// TIA Portal V20 export
TYPE "LER_typePLCToMotion"
// stored: Access Published
   STRUCT
      Commands : Struct
         Dancer : Struct
            Enable : Bool;
            Stop : Bool;
            Reset : Bool;
         END_STRUCT;
         StackMain : Struct
            Calculate : Bool;
            SemiStep : Bool;
            FullStep : Bool;
            Auto : Bool;
            SepaClean : Bool;
            CycleStop : Bool;
            FastStop : Bool;
            Reset : Bool;
         END_STRUCT;
      END_STRUCT;
      Parameters : Struct
         Dancer : Struct
            DancerDirection : Bool;
            UnWinderDirection : Bool;
            UnwinderTopUse : Bool;
            UnwinderBottomUse : Bool;
            Setpoint : LReal;
            Input : LReal;
            Kp : LReal;
            Ki : LReal;
            Radius : LReal;
            JogMode : Bool;
         END_STRUCT;
         StackMain : Struct
            Global : Struct
               CPM : LReal;
               StageWidth : LReal;
            END_STRUCT;
            "Step" : Struct
               MandrelUse : Bool;
               InitialPosFinalRoller : LReal;
               InitialPosCompensator : LReal;
            END_STRUCT;
            Auto : Struct
               SepaClean : Bool;
               CellCount : DInt;
               InitialPosFinalRoller : LReal;
               InitialPosCompensator : LReal;
               InitialPosAnodePnPX1 : LReal;
               InitialPosAnodePnPX2 : LReal;
               InitialPosAnodePnPZ1 : LReal;
               InitialPosAnodePnPZ2 : LReal;
               InitialPosCathodePnPX1 : LReal;
               InitialPosCathodePnPX2 : LReal;
               InitialPosCathodePnPZ1 : LReal;
               InitialPosCathodePnPZ2 : LReal;
               InitialPosAnodeMandrelYFront : LReal;
               InitialPosAnodeMandrelYRear : LReal;
               InitialPosAnodeMandrelZFront : LReal;
               InitialPosAnodeMandrelZRear : LReal;
               InitialPosCathodeMandrelYFront : LReal;
               InitialPosCathodeMandrelYRear : LReal;
               InitialPosCathodeMandrelZFront : LReal;
               InitialPosCathodeMandrelZRear : LReal;
               Pos1FinalRollerXFwdOutputCam : LReal;
               Pos1FinalRollerXBwdOutputCam : LReal;
               Pos1FinalRollerXStackTableDownOutputCam : LReal;
               Pos1FinalRollerXStackAnodeVisionOutputCam : LReal;
               Pos1FinalRollerXStackCathodeVisionOutputCam : LReal;
               Pos1AnodePnPX1FwdOutputCam : LReal;
               Pos1AnodePnPX1BwdOutputCam : LReal;
               Pos1AnodePnPX1ReelCutDataDeleteOffOutputCam : LReal;
               Pos1AnodePnPX2FwdOutputCam : LReal;
               Pos1AnodePnPX2BwdOutputCam : LReal;
               Pos1AnodePnPZ1Down1OutputCam : LReal;
               Pos1AnodePnPZ1Up1OutputCam : LReal;
               Pos1AnodePnPZ2Down1OutputCam : LReal;
               Pos1AnodePnPZ2Up1OutputCam : LReal;
               Pos1AnodePnPZ1Down2OutputCam : LReal;
               Pos1AnodePnPZ1Up2OutputCam : LReal;
               Pos1AnodePnPZ2Down2OutputCam : LReal;
               Pos1AnodePnPZ2Up2OutputCam : LReal;
               Pos1AnodePnPZ1SuctionOnOutputCam : LReal;
               Pos1AnodePnPZ1SuctionOffOutputCam : LReal;
               Pos1AnodePnPZ1ReelCutBlowOutputCam : LReal;
               Pos1AnodePnPZ1ReelCutDataDeleteOnOutputCam : LReal;
               Pos1AnodePnPZ1AlignVisionOutputCam : LReal;
               Pos1AnodePnPZ2SuctionOnOutputCam : LReal;
               Pos1AnodePnPZ2SuctionOffOutputCam : LReal;
               Pos1AnodeAlignSuctionOnOutputCam : LReal;
               Pos1AnodeAlignSuctionOffOutputCam : LReal;
               Pos1CathodePnPX1FwdOutputCam : LReal;
               Pos1CathodePnPX1BwdOutputCam : LReal;
               Pos1CathodePnPX1ReelCutDataDeleteOffOutputCam : LReal;
               Pos1CathodePnPX2FwdOutputCam : LReal;
               Pos1CathodePnPX2BwdOutputCam : LReal;
               Pos1CathodePnPZ1Down1OutputCam : LReal;
               Pos1CathodePnPZ1Up1OutputCam : LReal;
               Pos1CathodePnPZ2Down1OutputCam : LReal;
               Pos1CathodePnPZ2Up1OutputCam : LReal;
               Pos1CathodePnPZ1Down2OutputCam : LReal;
               Pos1CathodePnPZ1Up2OutputCam : LReal;
               Pos1CathodePnPZ2Down2OutputCam : LReal;
               Pos1CathodePnPZ2Up2OutputCam : LReal;
               Pos1CathodePnPZ1SuctionOnOutputCam : LReal;
               Pos1CathodePnPZ1SuctionOffOutputCam : LReal;
               Pos1CathodePnPZ1ReelCutBlowOutputCam : LReal;
               Pos1CathodePnPZ1ReelCutDataDeleteOnOutputCam : LReal;
               Pos1CathodePnPZ1AlignVisionOutputCam : LReal;
               Pos1CathodePnPZ2SuctionOnOutputCam : LReal;
               Pos1CathodePnPZ2SuctionOffOutputCam : LReal;
               Pos1CathodeAlignSuctionOnOutputCam : LReal;
               Pos1CathodeAlignSuctionOffOutputCam : LReal;
               Pos2FinalRollerXFwdOutputCam : LReal;
               Pos2FinalRollerXBwdOutputCam : LReal;
               Pos2FinalRollerXStackTableDownOutputCam : LReal;
               Pos2FinalRollerXStackAnodeVisionOutputCam : LReal;
               Pos2FinalRollerXStackCathodeVisionOutputCam : LReal;
               Pos2AnodePnPX1FwdOutputCam : LReal;
               Pos2AnodePnPX1BwdOutputCam : LReal;
               Pos2AnodePnPX1ReelCutDataDeleteOffOutputCam : LReal;
               Pos2AnodePnPX2FwdOutputCam : LReal;
               Pos2AnodePnPX2BwdOutputCam : LReal;
               Pos2AnodePnPZ1Down1OutputCam : LReal;
               Pos2AnodePnPZ1Up1OutputCam : LReal;
               Pos2AnodePnPZ2Down1OutputCam : LReal;
               Pos2AnodePnPZ2Up1OutputCam : LReal;
               Pos2AnodePnPZ1Down2OutputCam : LReal;
               Pos2AnodePnPZ1Up2OutputCam : LReal;
               Pos2AnodePnPZ2Down2OutputCam : LReal;
               Pos2AnodePnPZ2Up2OutputCam : LReal;
               Pos2AnodePnPZ1SuctionOnOutputCam : LReal;
               Pos2AnodePnPZ1SuctionOffOutputCam : LReal;
               Pos2AnodePnPZ1ReelCutBlowOutputCam : LReal;
               Pos2AnodePnPZ1ReelCutDataDeleteOnOutputCam : LReal;
               Pos2AnodePnPZ1AlignVisionOutputCam : LReal;
               Pos2AnodePnPZ2SuctionOnOutputCam : LReal;
               Pos2AnodePnPZ2SuctionOffOutputCam : LReal;
               Pos2AnodeAlignSuctionOnOutputCam : LReal;
               Pos2AnodeAlignSuctionOffOutputCam : LReal;
               Pos2CathodePnPX1FwdOutputCam : LReal;
               Pos2CathodePnPX1BwdOutputCam : LReal;
               Pos2CathodePnPX1ReelCutDataDeleteOffOutputCam : LReal;
               Pos2CathodePnPX2FwdOutputCam : LReal;
               Pos2CathodePnPX2BwdOutputCam : LReal;
               Pos2CathodePnPZ1Down1OutputCam : LReal;
               Pos2CathodePnPZ1Up1OutputCam : LReal;
               Pos2CathodePnPZ2Down1OutputCam : LReal;
               Pos2CathodePnPZ2Up1OutputCam : LReal;
               Pos2CathodePnPZ1Down2OutputCam : LReal;
               Pos2CathodePnPZ1Up2OutputCam : LReal;
               Pos2CathodePnPZ2Down2OutputCam : LReal;
               Pos2CathodePnPZ2Up2OutputCam : LReal;
               Pos2CathodePnPZ1SuctionOnOutputCam : LReal;
               Pos2CathodePnPZ1SuctionOffOutputCam : LReal;
               Pos2CathodePnPZ1ReelCutBlowOutputCam : LReal;
               Pos2CathodePnPZ1ReelCutDataDeleteOnOutputCam : LReal;
               Pos2CathodePnPZ1AlignVisionOutputCam : LReal;
               Pos2CathodePnPZ2SuctionOnOutputCam : LReal;
               Pos2CathodePnPZ2SuctionOffOutputCam : LReal;
               Pos2CathodeAlignSuctionOnOutputCam : LReal;
               Pos2CathodeAlignSuctionOffOutputCam : LReal;
            END_STRUCT;
            StackCalculate : Struct
               Direction : Bool := TRUE;
               RatioOption : Bool := TRUE;
               TimeOption : Bool;
               PosOption : Bool;
               DoubleOption : Bool;
               StageHeight : LReal := 360.0;
               StageGap : LReal := 5.0;
               AccRatio : DInt := 3;
               Ratio : Struct
                  FinalRollerStart : LReal := 0.0;
                  FinalRollerEnd : LReal := 75.0;
                  PnPXStart : LReal := 0.0;
                  PnPXEnd : LReal := 75.0;
                  PnPZDownStart : LReal := 65.0;
                  PnPZDownEnd : LReal := 75.0;
                  PnPZUpStart : LReal := 90.0;
                  PnPZUpEnd : LReal := 100.0;
                  MandrelBwdStart : LReal := 75.0;
                  MandrelBwdEnd : LReal := 82.5;
                  MandrelFwdStart : LReal := 82.5;
                  MandrelFwdEnd : LReal := 90.0;
                  MandrelUpStart1 : LReal := 55.0;
                  MandrelUpEnd1 : LReal := 62.5;
                  MandrelUpStart2 : LReal := 75.0;
                  MandrelUpEnd2 : LReal := 82.5;
                  MandrelDownStart : LReal := 87.0;
                  MandrelDownEnd : LReal := 90.0;
                  MandrelYTerm : LReal := 0.0;
                  MandrelZTerm : LReal := 0.0;
                  MandrelBwdOffset : LReal := 0.0;
                  MandrelFwdOffset : LReal := 0.0;
               END_STRUCT;
               "Time" : Struct
                  FinalRollerStart : LReal;
                  FinalRollerEnd : LReal;
                  PnPXStart : LReal;
                  PnPXEnd : LReal;
                  PnPZDownStart : LReal;
                  PnPZDownEnd : LReal;
                  PnPZUpStart : LReal;
                  PnPZUpEnd : LReal;
                  MandrelBwdStart : LReal;
                  MandrelBwdEnd : LReal;
                  MandrelFwdStart : LReal;
                  MandrelFwdEnd : LReal;
                  MandrelUpStart1 : LReal;
                  MandrelUpEnd1 : LReal;
                  MandrelUpStart2 : LReal;
                  MandrelUpEnd2 : LReal;
                  MandrelDownStart : LReal;
                  MandrelDownEnd : LReal;
               END_STRUCT;
               Position : Struct
                  FinalRollerBwdPos : LReal;
                  FinalRollerFwdPos : LReal;
               END_STRUCT;
               TeachingPos : Struct
                  StartPos : Struct
                     Compensator : LReal;
                     FinalRoller : LReal;
                     AnodePnPX1 : LReal;
                     AnodePnPX2 : LReal;
                     AnodePnPZ1 : LReal;
                     AnodePnPZ2 : LReal;
                     CathodePnPX1 : LReal;
                     CathodePnPX2 : LReal;
                     CathodePnPZ1 : LReal;
                     CathodePnPZ2 : LReal;
                     AnodeMandrelYFront : LReal;
                     AnodeMandrelYRear : LReal;
                     AnodeMandrelZFront : LReal;
                     AnodeMandrelZRear : LReal;
                     CathodeMandrelYFront : LReal;
                     CathodeMandrelYRear : LReal;
                     CathodeMandrelZFront : LReal;
                     CathodeMandrelZRear : LReal;
                  END_STRUCT;
                  EndPos : Struct
                     FinalRoller : LReal;
                     AnodePnPX1 : LReal;
                     AnodePnPX2 : LReal;
                     AnodePnPZ1P1 : LReal;
                     AnodePnPZ1P2 : LReal;
                     AnodePnPZ2P1 : LReal;
                     AnodePnPZ2P2 : LReal;
                     CathodePnPX1 : LReal;
                     CathodePnPX2 : LReal;
                     CathodePnPZ1P1 : LReal;
                     CathodePnPZ1P2 : LReal;
                     CathodePnPZ2P1 : LReal;
                     CathodePnPZ2P2 : LReal;
                     AnodeMandrelYFront : LReal;
                     AnodeMandrelYRear : LReal;
                     AnodeMandrelZFront : LReal;
                     AnodeMandrelZRear : LReal;
                     CathodeMandrelYFront : LReal;
                     CathodeMandrelYRear : LReal;
                     CathodeMandrelZFront : LReal;
                     CathodeMandrelZRear : LReal;
                  END_STRUCT;
               END_STRUCT;
            END_STRUCT;
         END_STRUCT;
      END_STRUCT;
      TechnologyObject : Struct
         Axis : Struct
            MasterVirtual : DB_ANY := 85;
            UnwinderVirtual : DB_ANY := 391;
            UnwinderTop : DB_ANY := 364;
            UnwinderBottom : DB_ANY := 263;
            FinalRoller : DB_ANY := 171;
            Compensator : DB_ANY := 143;
            AnodePnPX1 : DB_ANY := 144;
            AnodePnPX2 : DB_ANY := 145;
            AnodePnPZ1 : DB_ANY := 149;
            AnodePnPZ2 : DB_ANY := 150;
            CathodePnPX1 : DB_ANY := 146;
            CathodePnPX2 : DB_ANY := 147;
            CathodePnPZ1 : DB_ANY := 151;
            CathodePnPZ2 : DB_ANY := 153;
            AnodeMandrelYFront : DB_ANY := 163;
            AnodeMandrelYRear : DB_ANY := 162;
            AnodeMandrelZFront : DB_ANY := 167;
            AnodeMandrelZRear : DB_ANY := 166;
            CathodeMandrelYFront : DB_ANY := 161;
            CathodeMandrelYRear : DB_ANY := 160;
            CathodeMandrelZFront : DB_ANY := 165;
            CathodeMandrelZRear : DB_ANY := 164;
            SepaClampX : DB_ANY := 178;
         END_STRUCT;
         Cam : Struct
            FinalRollerCam { ExternalAccessible := 'False'; ExternalVisible := 'False'; ExternalWritable := 'False'} : DB_ANY := 281;
            CompensatorCam { ExternalAccessible := 'False'; ExternalVisible := 'False'; ExternalWritable := 'False'} : DB_ANY := 69;
            AnodePnPX1Cam { ExternalAccessible := 'False'; ExternalVisible := 'False'; ExternalWritable := 'False'} : DB_ANY := 230;
            AnodePnPX2Cam { ExternalAccessible := 'False'; ExternalVisible := 'False'; ExternalWritable := 'False'} : DB_ANY := 295;
            AnodePnPZ1Cam { ExternalAccessible := 'False'; ExternalVisible := 'False'; ExternalWritable := 'False'} : DB_ANY := 294;
            AnodePnPZ2Cam { ExternalAccessible := 'False'; ExternalVisible := 'False'; ExternalWritable := 'False'} : DB_ANY := 296;
            CathodePnPX1Cam { ExternalAccessible := 'False'; ExternalVisible := 'False'; ExternalWritable := 'False'} : DB_ANY := 293;
            CathodePnPX2Cam { ExternalAccessible := 'False'; ExternalVisible := 'False'; ExternalWritable := 'False'} : DB_ANY := 297;
            CathodePnPZ1Cam { ExternalAccessible := 'False'; ExternalVisible := 'False'; ExternalWritable := 'False'} : DB_ANY := 299;
            CathodePnPZ2Cam { ExternalAccessible := 'False'; ExternalVisible := 'False'; ExternalWritable := 'False'} : DB_ANY := 298;
            AnodeMandrelYFrontCam { ExternalAccessible := 'False'; ExternalVisible := 'False'; ExternalWritable := 'False'} : DB_ANY := 283;
            AnodeMandrelYRearCam { ExternalAccessible := 'False'; ExternalVisible := 'False'; ExternalWritable := 'False'} : DB_ANY := 285;
            AnodeMandrelZFrontCam { ExternalAccessible := 'False'; ExternalVisible := 'False'; ExternalWritable := 'False'} : DB_ANY := 287;
            AnodeMandrelZRearCam { ExternalAccessible := 'False'; ExternalVisible := 'False'; ExternalWritable := 'False'} : DB_ANY := 290;
            CathodeMandrelYFrontCam { ExternalAccessible := 'False'; ExternalVisible := 'False'; ExternalWritable := 'False'} : DB_ANY := 284;
            CathodeMandrelYRearCam { ExternalAccessible := 'False'; ExternalVisible := 'False'; ExternalWritable := 'False'} : DB_ANY := 289;
            CathodeMandrelZFrontCam { ExternalAccessible := 'False'; ExternalVisible := 'False'; ExternalWritable := 'False'} : DB_ANY := 286;
            CathodeMandrelZRearCam { ExternalAccessible := 'False'; ExternalVisible := 'False'; ExternalWritable := 'False'} : DB_ANY := 288;
         END_STRUCT;
         OutputCam : Struct
            FinalRollerXFwdOutputCam { ExternalAccessible := 'False'; ExternalVisible := 'False'; ExternalWritable := 'False'} : DB_ANY;
            FinalRollerXBwdOutputCam { ExternalAccessible := 'False'; ExternalVisible := 'False'; ExternalWritable := 'False'} : DB_ANY;
            FinalRollerXStackTableDownOutputCam { ExternalAccessible := 'False'; ExternalVisible := 'False'; ExternalWritable := 'False'} : DB_ANY;
            FinalRollerXStackAnodeVisionOutputCam { ExternalAccessible := 'False'; ExternalVisible := 'False'; ExternalWritable := 'False'} : DB_ANY;
            FinalRollerXStackCathodeVisionOutputCam { ExternalAccessible := 'False'; ExternalVisible := 'False'; ExternalWritable := 'False'} : DB_ANY;
            AnodePnPX1FwdOutputCam { ExternalAccessible := 'False'; ExternalVisible := 'False'; ExternalWritable := 'False'} : DB_ANY;
            AnodePnPX1BwdOutputCam { ExternalAccessible := 'False'; ExternalVisible := 'False'; ExternalWritable := 'False'} : DB_ANY;
            AnodePnPX2FwdOutputCam { ExternalAccessible := 'False'; ExternalVisible := 'False'; ExternalWritable := 'False'} : DB_ANY;
            AnodePnPX2BwdOutputCam { ExternalAccessible := 'False'; ExternalVisible := 'False'; ExternalWritable := 'False'} : DB_ANY;
            AnodePnPZ1Down1OutputCam { ExternalAccessible := 'False'; ExternalVisible := 'False'; ExternalWritable := 'False'} : DB_ANY;
            AnodePnPZ1Up1OutputCam { ExternalAccessible := 'False'; ExternalVisible := 'False'; ExternalWritable := 'False'} : DB_ANY;
            AnodePnPZ2Down1OutputCam { ExternalAccessible := 'False'; ExternalVisible := 'False'; ExternalWritable := 'False'} : DB_ANY;
            AnodePnPZ2Up1OutputCam { ExternalAccessible := 'False'; ExternalVisible := 'False'; ExternalWritable := 'False'} : DB_ANY;
            AnodePnPZ1Down2OutputCam { ExternalAccessible := 'False'; ExternalVisible := 'False'; ExternalWritable := 'False'} : DB_ANY;
            AnodePnPZ1Up2OutputCam { ExternalAccessible := 'False'; ExternalVisible := 'False'; ExternalWritable := 'False'} : DB_ANY;
            AnodePnPZ2Down2OutputCam { ExternalAccessible := 'False'; ExternalVisible := 'False'; ExternalWritable := 'False'} : DB_ANY;
            AnodePnPZ2Up2OutputCam { ExternalAccessible := 'False'; ExternalVisible := 'False'; ExternalWritable := 'False'} : DB_ANY;
            AnodePnPZ1SuctionOnOutputCam { ExternalAccessible := 'False'; ExternalVisible := 'False'; ExternalWritable := 'False'} : DB_ANY;
            AnodePnPZ1SuctionOffOutputCam { ExternalAccessible := 'False'; ExternalVisible := 'False'; ExternalWritable := 'False'} : DB_ANY;
            AnodePnPZ1ReelCutBlowOutputCam { ExternalAccessible := 'False'; ExternalVisible := 'False'; ExternalWritable := 'False'} : DB_ANY;
            AnodePnPZ2SuctionOnOutputCam { ExternalAccessible := 'False'; ExternalVisible := 'False'; ExternalWritable := 'False'} : DB_ANY;
            AnodePnPZ2SuctionOffOutputCam { ExternalAccessible := 'False'; ExternalVisible := 'False'; ExternalWritable := 'False'} : DB_ANY;
            AnodeAlignSuctionOnOutputCam { ExternalAccessible := 'False'; ExternalVisible := 'False'; ExternalWritable := 'False'} : DB_ANY;
            AnodeAlignSuctionOffOutputCam { ExternalAccessible := 'False'; ExternalVisible := 'False'; ExternalWritable := 'False'} : DB_ANY;
            AnodePnPZ1ReelCutDataDeleteOnOutputCam { ExternalAccessible := 'False'; ExternalVisible := 'False'; ExternalWritable := 'False'} : DB_ANY;
            AnodePnP1XReelCutDataDeleteOffOutputCam { ExternalAccessible := 'False'; ExternalVisible := 'False'; ExternalWritable := 'False'} : DB_ANY;
            AnodeAlignVisionOutputCam { ExternalAccessible := 'False'; ExternalVisible := 'False'; ExternalWritable := 'False'} : DB_ANY;
            CathodePnPX1FwdOutputCam { ExternalAccessible := 'False'; ExternalVisible := 'False'; ExternalWritable := 'False'} : DB_ANY;
            CathodePnPX1BwdOutputCam { ExternalAccessible := 'False'; ExternalVisible := 'False'; ExternalWritable := 'False'} : DB_ANY;
            CathodePnPX2FwdOutputCam { ExternalAccessible := 'False'; ExternalVisible := 'False'; ExternalWritable := 'False'} : DB_ANY;
            CathodePnPX2BwdOutputCam { ExternalAccessible := 'False'; ExternalVisible := 'False'; ExternalWritable := 'False'} : DB_ANY;
            CathodePnPZ1Down1OutputCam { ExternalAccessible := 'False'; ExternalVisible := 'False'; ExternalWritable := 'False'} : DB_ANY;
            CathodePnPZ1Up1OutputCam { ExternalAccessible := 'False'; ExternalVisible := 'False'; ExternalWritable := 'False'} : DB_ANY;
            CathodePnPZ2Down1OutputCam { ExternalAccessible := 'False'; ExternalVisible := 'False'; ExternalWritable := 'False'} : DB_ANY;
            CathodePnPZ2Up1OutputCam { ExternalAccessible := 'False'; ExternalVisible := 'False'; ExternalWritable := 'False'} : DB_ANY;
            CathodePnPZ1Down2OutputCam { ExternalAccessible := 'False'; ExternalVisible := 'False'; ExternalWritable := 'False'} : DB_ANY;
            CathodePnPZ1Up2OutputCam { ExternalAccessible := 'False'; ExternalVisible := 'False'; ExternalWritable := 'False'} : DB_ANY;
            CathodePnPZ2Down2OutputCam { ExternalAccessible := 'False'; ExternalVisible := 'False'; ExternalWritable := 'False'} : DB_ANY;
            CathodePnPZ2Up2OutputCam { ExternalAccessible := 'False'; ExternalVisible := 'False'; ExternalWritable := 'False'} : DB_ANY;
            CathodePnPZ1SuctionOnOutputCam { ExternalAccessible := 'False'; ExternalVisible := 'False'; ExternalWritable := 'False'} : DB_ANY;
            CathodePnPZ1SuctionOffOutputCam { ExternalAccessible := 'False'; ExternalVisible := 'False'; ExternalWritable := 'False'} : DB_ANY;
            CathodePnPZ1ReelCutBlowOutputCam { ExternalAccessible := 'False'; ExternalVisible := 'False'; ExternalWritable := 'False'} : DB_ANY;
            CathodePnPZ2SuctionOnOutputCam { ExternalAccessible := 'False'; ExternalVisible := 'False'; ExternalWritable := 'False'} : DB_ANY;
            CathodePnPZ2SuctionOffOutputCam { ExternalAccessible := 'False'; ExternalVisible := 'False'; ExternalWritable := 'False'} : DB_ANY;
            CathodeAlignSuctionOnOutputCam { ExternalAccessible := 'False'; ExternalVisible := 'False'; ExternalWritable := 'False'} : DB_ANY;
            CathodeAlignSuctionOffOutputCam { ExternalAccessible := 'False'; ExternalVisible := 'False'; ExternalWritable := 'False'} : DB_ANY;
            CathodePnPZ1ReelCutDataDeleteOnOutputCam { ExternalAccessible := 'False'; ExternalVisible := 'False'; ExternalWritable := 'False'} : DB_ANY;
            CathodePnP1XReelCutDataDeleteOffOutputCam { ExternalAccessible := 'False'; ExternalVisible := 'False'; ExternalWritable := 'False'} : DB_ANY;
            CathodeAlignVisionOutputCam { ExternalAccessible := 'False'; ExternalVisible := 'False'; ExternalWritable := 'False'} : DB_ANY;
         END_STRUCT;
      END_STRUCT;
      Interface : Struct
         AnodeReelcutStandby : Bool;
         CathodeReelcutStandby : Bool;
         AnodeReelcutDone : Bool;
         CathodeReelcutDone : Bool;
      END_STRUCT;
   END_STRUCT;
END_TYPE
